// TIA Portal V20 export
ORGANIZATION_BLOCK "Main"   // OB1031, LAD, ProgramCycle
TITLE = "Main Program Sweep (Cycle)"
AUTHOR : ERsystem_FA2_DH. Kim
// stored: AutoNumber false, IsIECCheckEnabled true, Namespace Unit1.Em3, SetENOAutomatically false
   VAR_INPUT
      Initial_Call : Bool;   // Initial call of this OB
      Remanence : Bool;   // =True, if remanent data are available
   END_VAR
   VAR_TEMP
      tempIndex : Int;   // Index of EM in the array
   END_VAR
BEGIN

REGION Network 1: Call Simulation
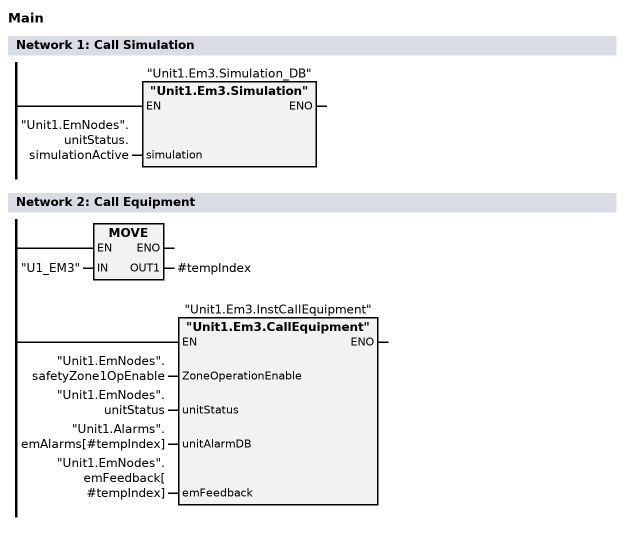
   RUNG wire#powerrail
      "Unit1.Em3.Simulation_DB"(simulation := "Unit1.EmNodes".unitStatus.simulationActive)
   END_RUNG
   // the same network as SCL:
   "Unit1.Em3.Simulation_DB"(simulation := "Unit1.EmNodes".unitStatus.simulationActive);   // "Unit1.Em3.Simulation"
END_REGION

REGION Network 2: Call Equipment
   RUNG wire#powerrail
      Move(in := "U1_EM3", out1 => #tempIndex)
   END_RUNG
   RUNG wire#powerrail
      "Unit1.Em3.InstCallEquipment"(ZoneOperationEnable := "Unit1.EmNodes".safetyZone1OpEnable, unitStatus := "Unit1.EmNodes".unitStatus, unitAlarmDB := "Unit1.Alarms".emAlarms[#tempIndex], emFeedback := "Unit1.EmNodes".emFeedback[#tempIndex])
   END_RUNG
   // the same network as SCL:
   #tempIndex := "U1_EM3";
   "Unit1.Em3.InstCallEquipment"(ZoneOperationEnable := "Unit1.EmNodes".safetyZone1OpEnable,   // "Unit1.Em3.CallEquipment"
                           unitStatus := "Unit1.EmNodes".unitStatus,
                           unitAlarmDB := "Unit1.Alarms".emAlarms[#tempIndex],
                           emFeedback := "Unit1.EmNodes".emFeedback[#tempIndex]);
END_REGION
END_ORGANIZATION_BLOCK
